{attribute 'GeneratedUsingTerminal: EL6614-0000-0016'}
{attribute addProperty BoxType "EL6614-0000-0016"}
{attribute addProperty Id "EtcSlaveTerminalBaseInfoDataAT %I*InfoData_32EB74EA10"}
{attribute addProperty CRC "3667650902"}
{attribute addProperty Size "10"}
TYPE EL6614_DA9BE956 EXTENDS EtcSlaveTerminalBase :
STRUCT
	{attribute addProperty Name "InfoData"}
	InfoData : InfoData_32EB74EA;
END_STRUCT
END_TYPE

(* stored: Version 1.2.0.0, ProductVersion 3.1.4024.9
   DUT EL6614_DA9BE956: Id {03847f1a-518e-4f97-a56b-94a5046c0c02} *)
